KUKA KRL program: style1app2opt2.src, style1app2opt2.dat

--- style1app2opt2.src ---
&ACCESS RVO1
&REL 16
&COMMENT 03-10-R1 NUT CHECK CAMERA
&PARAM EDITMASK = *
&PARAM DISKPATH = KRC:\R1\Program\StyleApps\Options
DEF Style1App2Opt2( )
   ;FOLD INI
      ;FOLD BASISTECH INI
         GLOBAL INTERRUPT DECL 3 WHEN $STOPMESS==TRUE DO IR_STOPM ( )
         INTERRUPT ON 3
         BAS (#INITMOV,0 )
      ;ENDFOLD (BASISTECH INI)
      ;FOLD USER INI
         ;Make your modifications here

      ;ENDFOLD (USER INI)
   ;ENDFOLD (INI)
;********************************
; Gestamp Standards
; Line - BMW G65 (cell 03)
; Robot 03-10-R1 (BMW-03-10-R1-MH1)
; Application - NUT CHECK WITH THE CAMERA
;********************************
; CALLED BY Style1Opt1 AND Style1Opt10AutoRR AFTER THE SENSOR CHECK (style1app2opt1).
; PRESENTS THE PART TO THE CAMERA (P3), ASKS THE PLC FOR THE INSPECTION ($OUT[80]) AND SETS
; bscrapGE4 FROM THE RESULT; THEN RELEASES APPLICATION 1.
;NOTE: THE CAMERA RESULT IS EVALUATED BY OPTION (PRODUCTION 1, 2, 7, 8; RED RABBIT 12), ALSO IN
;  DRY CYCLE (F02, F05, F19)
;APPROACH THE CAMERA - P6 (TAUGHT IN BASE 3 "NUT WELDER")
;FOLD PTP P6 Vel=100 % PDAT10 Tool[1]:TOOL 1 Base[3]:NUT WELDER;%{PE}%R 8.3.43,%MKUKATPBASIS,%CMOVE,%VPTP,%P 1:PTP, 2:P6, 3:, 5:100, 7:PDAT10
$BWDSTART=FALSE
PDAT_ACT=PPDAT10
FDAT_ACT=FP6
BAS(#PTP_PARAMS,100)
PTP XP6
;ENDFOLD

;PART AT THE CAMERA - LIN P3 (1 M/S, EXACT STOP)
;FOLD LIN P3 Vel=1 m/s CPDAT0 Tool[1]:TOOL 1 Base[0];%{PE}%R 8.3.43,%MKUKATPBASIS,%CMOVE,%VLIN,%P 1:LIN, 2:P3, 3:, 5:1, 7:CPDAT0
$BWDSTART=FALSE
LDAT_ACT=LCPDAT0
FDAT_ACT=FP3
BAS(#CP_PARAMS,1)
LIN XP3
;ENDFOLD

;CAMERA INSPECTION REQUEST - SIGNAL $OUT[80] do080RepositionTooling1 ON
;NOTE: NOTHING IN THE PROGRAM SWITCHES $OUT[80] OFF AGAIN (ONLY MaintainSystem AT THE NEXT CYCLE
;  START): THE PLC MAY SEE A STANDING REQUEST WHILE THE ROBOT LEAVES (F15)
do080RepositionTooling1=TRUE

;WAIT INSPECTION DONE - SIGNAL $IN[80] di080ToolRepositioned1 ON (NO TIMEOUT, F15)
   WAIT FOR di080ToolRepositioned1

;AFTER 0.2 S, BY OPTION nOption (F02, F19):
;PRODUCTION OPTIONS 1, 2, 7, 8: GOOD (bscrapGE4 = FALSE) ONLY WITH $IN[100] di100CameraJudgmentOK ON
;AND $IN[101] di101CameraJudgmentNG OFF; NG OR NO VALID RESULT -> bscrapGE4 = TRUE (SCRAP)
;RED RABBIT OPTION 12: CAMERA OK -> $OUT[141] do141RedRabbitFailed ON; CAMERA NG ->
;$OUT[142] do142RedRabbitPassed ON
            WAIT SEC 0.2
     SWITCH nOption
          CASE 1,2,7,8
         ;GOOD - SIGNALS $IN[100] di100CameraJudgmentOK ON, $IN[101] di101CameraJudgmentNG OFF
         IF (di100CameraJudgmentOK==TRUE) AND (di101CameraJudgmentNG==FALSE) THEN
            bscrapGE4 = FALSE
         ELSE
            bscrapGE4 = TRUE
         ENDIF
          CASE 12
         ;RED RABBIT FAILED - $IN[100] di100CameraJudgmentOK ON, $IN[101] di101CameraJudgmentNG OFF:
         ;SIGNAL $OUT[141] do141RedRabbitFailed ON
         IF (di100CameraJudgmentOK==TRUE) AND (di101CameraJudgmentNG==FALSE) THEN
            do141RedRabbitFailed=TRUE
         ENDIF
         ;RED RABBIT PASSED - $IN[100] di100CameraJudgmentOK OFF, $IN[101] di101CameraJudgmentNG ON:
         ;SIGNAL $OUT[142] do142RedRabbitPassed ON
         IF (di100CameraJudgmentOK==FALSE) AND (di101CameraJudgmentNG==TRUE) THEN
            do142RedRabbitPassed=TRUE
         ENDIF
     ENDSWITCH


;APPLICATION 1 CLEAR - AC_Application(1,TRUE): SIGNAL $OUT[70] do070ApplicationClear1 ON
;WARNING: HIDDEN AC_CmdParam=2 - CONFIRMING THIS FORM REGENERATES AC_Application(2,TRUE) (F21)
;NOTE: A SCRAP DECIDED BY THE SENSOR CHECK SKIPS THIS PROGRAM: APPLICATION 1 IS THEN NOT
;  RELEASED BY THE ROBOT (F20)
   ;FOLD Application[1] Reset
      ;FOLD ;%{h}
         ;Params IlfProvider=ac_zoneilf; AC_CmdZones=Application; AC_CmdParam=2; AC_ZoneRepo=True; AC_Blending=False
      ;ENDFOLD
      AC_Application (1,True)
   ;ENDFOLD
END

--- style1app2opt2.dat ---
&ACCESS RVO1
&REL 16
&COMMENT GE4_NutCHK
&PARAM EDITMASK = *
&PARAM DISKPATH = KRC:\R1\Program\StyleApps\Options
DEFDAT  Style1App2Opt2
;FOLD EXTERNAL DECLARATIONS;%{PE}%MKUKATPBASIS,%CEXT,%VCOMMON,%P
;FOLD BASISTECH EXT;%{PE}%MKUKATPBASIS,%CEXT,%VEXT,%P
EXT  BAS (BAS_COMMAND  :IN,REAL  :IN )
;ENDFOLD (BASISTECH EXT)
;FOLD USER EXT;%{E}%MKUKATPUSER,%CEXT,%VEXT,%P
;Make here your modifications
;ENDFOLD (USER EXT)
;ENDFOLD (EXTERNAL DECLARATIONS)
DECL BASIS_SUGG_T LAST_BASIS={POINT1[] "P0                      ",POINT2[] "P0                      ",CP_PARAMS[] "CPDAT0                  ",PTP_PARAMS[] "PDAT0                   ",CONT[] "                        ",CP_VEL[] "2.0                     ",PTP_VEL[] " 100                    ",SYNC_PARAMS[] "SYNCDAT                 ",SPL_NAME[] "S0                      ",A_PARAMS[] "ADAT0                   "}

DECL LDAT LCPDAT0={VEL 2.00000,ACC 80.0000,APO_DIST 100.000,APO_FAC 50.0000,AXIS_VEL 100.000,AXIS_ACC 100.000,ORI_TYP #VAR,CIRC_TYP #BASE,JERK_FAC 50.0000,GEAR_JERK 50.0000,EXAX_IGN 0}
DECL E6POS XP3={X -709.833740,Y -2035.40430,Z 1423.71777,A -98.4577484,B -5.84655905,C -164.806564,S 2,T 34,E1 0.0,E2 0.0,E3 0.0,E4 0.0,E5 0.0,E6 0.0}
DECL FDAT FP3={TOOL_NO 1,BASE_NO 0,IPO_FRAME #BASE,POINT2[] " ",TQ_STATE FALSE}
DECL E6POS XP6={X -3780.88599,Y -731.523132,Z -847.811157,A -165.231735,B -0.613393545,C -0.0522668548,S 2,T 34,E1 0.0,E2 0.0,E3 0.0,E4 0.0,E5 0.0,E6 0.0}
DECL FDAT FP6={TOOL_NO 1,BASE_NO 3,IPO_FRAME #BASE,POINT2[] " ",TQ_STATE FALSE}
DECL PDAT PPDAT10={VEL 100.000,ACC 100.000,APO_DIST 100.000,APO_MODE #CDIS,GEAR_JERK 50.0000,EXAX_IGN 0}
ENDDAT
